TYPE NodeId : DINT; END_TYPE

(* stored: Version 1.1.0.1, ProductVersion 3.1.4024.12
   DUT NodeId: Id {15518585-1b84-0de1-011f-7d84c8d47125} *)
